TYPE ST_TransportTubeOps :
STRUCT
	// Pumps
	bIonPumpIgnore : BOOL;
	
	// Valves
	bGateValveIgnore : BOOL;
	
	// Gauges
	ePiraniOp : E_GaugeCompOp;
	eColdCathodeOp : E_GaugeCompOp;
END_STRUCT
END_TYPE

(* stored: Version 1.1.0.1, ProductVersion 3.1.4024.0
   DUT ST_TransportTubeOps: Id {ec52e162-4e74-013e-040f-0be8b0b5fc20} *)
